PROGRAM IRTRANS_DEMO
VAR
	IP_C : IP_C;
	S_BUF : NETWORK_BUFFER_SHORT;
	R_BUF : NETWORK_BUFFER_SHORT;
	IP_CONTROL2 : IP_CONTROL2;
	IRTRANS_DECODE : IRTRANS_DECODE;
	IRTRANS_RCV_4 : IRTRANS_RCV_4;
	DRIVER_4 : DRIVER_4;
	IRTRANS_SERVER : IRTRANS_SERVER;
	IRTRANS_SND_8_1 : IRTRANS_SND_8;
	IRTRANS_SND_8_2 : IRTRANS_SND_8;
	Q0: BOOL;
	Q1: BOOL;
	Q2: BOOL;
	Q3: BOOL;
	error: BOOL;
	error_server: DWORD;
	Send_1_0: BOOL := TRUE;
	Send_1_1: BOOL;
	Send_1_2: BOOL;
	Send_1_3: BOOL;
	Send_1_4: BOOL;
	Send_1_5: BOOL;
	Send_1_6: BOOL;
	Send_1_7: BOOL;
	Send_2_0: BOOL := TRUE;
	Send_2_1: BOOL;
	Send_2_2: BOOL;
	Send_2_3: BOOL;
	Send_2_4: BOOL;
	Send_2_5: BOOL;
	Send_2_6: BOOL;
	Send_2_7: BOOL;
	R_ENABLE: BOOL;
	S_ENABLE: BOOL;
	MODE: BOOL := FALSE;
	KEY_1: BYTE;
	KEY_2: BYTE;
END_VAR

// note: 21 stored wires end on pins the file does not list and are not shown
// IRTRANS Empfang
IRTRANS_DECODE(IP_C := IP_C, R_BUF := R_BUF);
error := IRTRANS_DECODE.ERROR;
IRTRANS_RCV_4();
DRIVER_4(
    _in2 := IRTRANS_RCV_4.Q0,
    _in3 := IRTRANS_RCV_4.Q1,
    _in4 := IRTRANS_RCV_4.Q2,
    _in5 := IRTRANS_RCV_4.Q3);
Q0 := DRIVER_4._out1;
Q1 := DRIVER_4._out2;
Q2 := DRIVER_4._out3;
Q3 := DRIVER_4._out4;
// IRTRANS Senden (beliebig viele Instanzen zulässig !)
IRTRANS_SND_8_1(IN_0 := IP_C, IN_1 := S_BUF); // IRTRANS_SND_8
KEY_1 := IRTRANS_SND_8_1.KEY;
IRTRANS_SND_8_2(IN_0 := IP_C, IN_1 := S_BUF); // IRTRANS_SND_8
KEY_2 := IRTRANS_SND_8_2.KEY;
// IRTRANS Kommunikation
IRTRANS_SERVER(UDP_TCP := MODE, IP_C := IP_C, S_BUF := S_BUF, R_BUF := R_BUF);
S_ENABLE := IRTRANS_SERVER.S_ENABLE;
R_ENABLE := IRTRANS_SERVER.R_ENABLE;
error_server := IRTRANS_SERVER.ERROR;
// Hardwareneutraler Ethernet IP
IP_CONTROL2(PORT := 21000, TIME_OUT := T#2s, IP_C := IP_C, S_BUF := S_BUF, R_BUF := R_BUF);
// Send_1_0: input not connected
// Send_1_1: input not connected
// Send_1_2: input not connected
// Send_1_3: input not connected
// Send_1_4: input not connected
// Send_1_5: input not connected
// Send_1_6: input not connected
// Send_1_7: input not connected
// Send_2_0: input not connected
// Send_2_1: input not connected
// Send_2_2: input not connected
// Send_2_3: input not connected
// Send_2_4: input not connected
// Send_2_5: input not connected
// Send_2_6: input not connected
// Send_2_7: input not connected
// T#500ms: input not connected
// T#500ms: input not connected

END_PROGRAM

(* stored: Version 1.1.0.1, ProductVersion 3.1.4024.9
   POU IRTRANS_DEMO: Id {9ebeec48-185b-4726-b957-ace0ae1d4729}, SpecialFunc None *)
